(* IEC 61131-3 sources: Industrial-Meter-Tracking-System-Modernization/plc/function-blocks, 3 files *)

(* ---- calc-delta-t-fb.st ---- *)
(*
    Function Block: CalcDeltaT
    Purpose:
    Measures pulse duration from a digital sensor.

    Description:
    This block detects rising and falling edges of a sensor signal.
    On rising edge, it stores the start time.
    On falling edge, it calculates pulse duration.

    It stores minimum and maximum pulse duration within configured limits.

    Note:
    This is an anonymized version of the original industrial PLC logic.
*)

FUNCTION_BLOCK CalcDeltaT

VAR_INPUT
    Sensor   : BOOL;
    Reset    : BOOL;
    MAX_T_ms : UDINT;
    MIN_T_ms : UDINT;
END_VAR

VAR_OUTPUT
    MinTime : UDINT;
    MaxTime : UDINT;
END_VAR

VAR
    StartTimeMs : UDINT;
    PulseTimeMs : UDINT;

    RisingEdge  : BOOL;
    FallingEdge : BOOL;

    FirstRun    : BOOL;
    SensorPrev  : BOOL;
END_VAR

// Initialization or reset
IF (NOT FirstRun) OR Reset THEN
    FirstRun := TRUE;
    MaxTime := MIN_T_ms;
    MinTime := MAX_T_ms;
END_IF;

// Rising edge detection
IF (SensorPrev = FALSE) AND (Sensor = TRUE) THEN
    RisingEdge := TRUE;
ELSE
    RisingEdge := FALSE;
END_IF;

// Falling edge detection
IF (SensorPrev = TRUE) AND (Sensor = FALSE) THEN
    FallingEdge := TRUE;
ELSE
    FallingEdge := FALSE;
END_IF;

// Save pulse start time
IF RisingEdge THEN
    StartTimeMs := SysTimeRtc.SysTimeGetMs();
END_IF;

// Calculate pulse duration
IF FallingEdge THEN
    PulseTimeMs := SysTimeRtc.SysTimeGetMs() - StartTimeMs;

    IF (PulseTimeMs > MaxTime) AND (PulseTimeMs < MAX_T_ms) THEN
        MaxTime := PulseTimeMs;
    END_IF;

    IF (PulseTimeMs < MinTime) AND (PulseTimeMs > MIN_T_ms) THEN
        MinTime := PulseTimeMs;
    END_IF;
END_IF;

// Store previous sensor state
SensorPrev := Sensor;

(* ---- cut-point-fb.st ---- *)
(*
    Function Block: CutPoint
    Purpose:
    Detects counter reset event and captures last valid meter value.

    Description:
    This block processes incoming meter values from a counter.
    When a reset event is detected (sudden drop), it stores the last
    valid value before reset and signals that data is ready for transfer.

    Outputs:
    - AllMeters  : current valid value
    - AllMeters2 : value prepared for sending (buffer)
    - AllMeters3 : previous sent value (history)

    Notes:
    - Uses filtering to ignore invalid/overflow values
    - Designed for industrial environment with noisy signals
*)

FUNCTION_BLOCK CutPoint

VAR_INPUT
    Meters : DWORD;
END_VAR

VAR_IN_OUT
    Set : WORD; // signal for SCADA / WinCC
END_VAR

VAR_OUTPUT
    AllMeters  : DWORD; // current valid value
    AllMeters2 : DWORD; // buffer for transfer
    AllMeters3 : DWORD; // previous transferred value
END_VAR

VAR
    PrevMeters    : DWORD := 0;
    CurrMeters    : DWORD := 0;
    InitDone      : BOOL := FALSE;
    ResetDetected : BOOL := FALSE;

    MinDrop    : DWORD := 300;     // reset detection threshold (~30 m)
    ResetLevel : DWORD := 100;     // value after reset (~10 m)
    MaxValid   : DWORD := 1000000; // overflow filter

    ValidValue : BOOL := FALSE;
END_VAR

// --- Validate incoming value ---
IF Meters <= MaxValid THEN
    CurrMeters := Meters;
    ValidValue := TRUE;
ELSE
    ValidValue := FALSE;
END_IF;

// --- Initialization ---
IF (NOT InitDone) AND ValidValue THEN
    PrevMeters := CurrMeters;
    AllMeters := CurrMeters;
    InitDone := TRUE;
END_IF;

// --- Main logic ---
IF InitDone AND ValidValue THEN

    // Update current value
    AllMeters := CurrMeters;

    // Detect reset event
    IF (NOT ResetDetected)
       AND (PrevMeters > CurrMeters)
       AND ((PrevMeters - CurrMeters) > MinDrop)
       AND (CurrMeters < ResetLevel) THEN

        // Shift history
        AllMeters3 := AllMeters2;

        // Store last valid value before reset
        AllMeters2 := PrevMeters;

        // Signal SCADA
        Set := 1;

        ResetDetected := TRUE;
    END_IF;

    // Allow next reset detection when value increases
    IF CurrMeters > PrevMeters THEN
        ResetDetected := FALSE;
    END_IF;

    // Update previous value
    PrevMeters := CurrMeters;

END_IF;

(* ---- mb-reset-fb.st ---- *)
(*
    Function Block: MB_Reset
    Purpose:
    Handles automatic recovery of Modbus communication.

    Description:
    This block monitors communication errors and attempts to reset
    the Modbus channel when repeated failures occur.

    Logic:
    - If error persists → trigger reset periodically
    - Count number of reset attempts
    - If too many attempts → mark device as disconnected

    Notes:
    - Designed for industrial environment with unstable RS-485
*)

FUNCTION_BLOCK MB_Reset

VAR_INPUT
    Error        : BOOL; // communication error
    Done         : BOOL; // operation completed
    OutDone      : BOOL; // external completion signal
    ResetCommand : BOOL; // manual reset command
END_VAR

VAR_OUTPUT
    Reset            : BOOL; // reset signal to device
    DeviceLost       : BOOL; // device considered disconnected
END_VAR

VAR
    DoneInternal     : BOOL;
    ResetAttempts    : WORD;

    ErrorTimer       : TON;
    NoErrorTimer     : TON;

    RisingEdge       : R_TRIG;
END_VAR

// --- Determine internal "Done" state ---
IF (NOT OutDone) THEN
    DoneInternal := Done;
ELSE
    // wait until no error for 1 minute
    NoErrorTimer(IN := NOT Error, PT := T#1M, Q => DoneInternal);
END_IF;

// --- Reset state if communication restored or manual reset ---
IF ((DoneInternal AND (NOT Error)) OR ResetCommand) THEN
    ResetAttempts := 0;
    DeviceLost := FALSE;
    Reset := FALSE;
END_IF;

// --- If error present, keep reset off until timer triggers ---
IF Error THEN
    Reset := FALSE;
END_IF;

// --- Trigger reset every 3 seconds while error persists ---
ErrorTimer(IN := Error AND NOT ErrorTimer.Q, PT := T#3S);

RisingEdge(CLK := ErrorTimer.Q);

IF RisingEdge.Q THEN
    ResetAttempts := ResetAttempts + 1;
    Reset := TRUE;
END_IF;

// --- If too many attempts → mark device as lost ---
IF (ResetAttempts > 120) THEN
    Reset := FALSE;
    DeviceLost := TRUE;
END_IF;
